// TIA Portal V17 export
// export: Created 2022-07-20T07:01:31.1393195Z, ExportSetting WithDefaults, DisplayName Totally Integrated Automation Portal, DisplayVersion V17, DisplayName TIA Portal Openness, DisplayVersion V17, DisplayName TIA Portal Version Control Interface, DisplayVersion V17, DisplayName SINAMICS Startdrive Advanced, DisplayVersion V17, DisplayName SINAMICS Startdrive G130, G150, S120, S150, SINAMICS MV, S210, DisplayVersion V17, DisplayName SINAMICS Startdrive G110M, G120, G120C, G120D, G120P, G115D, DisplayVersion V17, DisplayName STEP 7 Professional, DisplayVersion V17, DisplayName STEP 7 Safety, DisplayVersion V17, DisplayName WinCC Advanced, DisplayVersion V17
FUNCTION_BLOCK "FB10041_DetectKindOfPush"   // FB10041, LAD
{ S7_Optimized_Access := 'TRUE' }
VERSION : 0.1
// stored: AutoNumber false, IsIECCheckEnabled false, IsRetainMemResEnabled false, MemoryReserve 100, SetENOAutomatically false, UDAEnableTagReadback false
   VAR_INPUT
      Push : Bool;
   END_VAR
   VAR_OUTPUT
      ShortPushDetected : Bool;
      LongPushDetected : Bool;
   END_VAR
   VAR
      ResetCounter : Bool;
      R_TRIG_Push : R_TRIG;
      F_TRIG_Push : F_TRIG;
      FB10220_OperatingTimeCounter_Instance { S7_SetPoint := 'True'} : "FB10220_OperatingTimeCounter";
   END_VAR
BEGIN

REGION Network 1 (SCL): First Scan
   IF "FirstScan" THEN
       #ShortPushDetected := FALSE;
       #LongPushDetected := FALSE;
   END_IF;
END_REGION

REGION Network 2 (SCL)
   REGION EDGE SIGNALS
       #R_TRIG_Push(CLK := #Push);

       #F_TRIG_Push(CLK := #Push);
   END_REGION
END_REGION

REGION Network 3: Push Counter Management
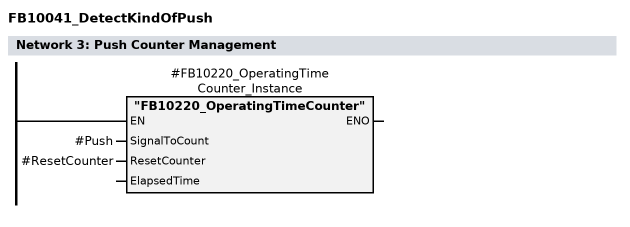
   RUNG wire#powerrail
      #FB10220_OperatingTimeCounter_Instance(SignalToCount := #Push, ResetCounter := #ResetCounter, ElapsedTime :=)
   END_RUNG
   // the same network as SCL:
   #FB10220_OperatingTimeCounter_Instance(SignalToCount := #Push, ResetCounter := #ResetCounter);   // "FB10220_OperatingTimeCounter"
END_REGION

REGION Network 4 (SCL): Kind Of Push Detection Management
   IF #R_TRIG_Push.Q THEN
       #ResetCounter := TRUE;
       #ShortPushDetected := FALSE;
       #LongPushDetected := FALSE;
   ELSIF #Push AND #FB10220_OperatingTimeCounter_Instance.ElapsedTime >= 1.0 THEN
       #ResetCounter := FALSE;
       #ShortPushDetected := FALSE;
       #LongPushDetected := TRUE;
   ELSIF #F_TRIG_Push.Q THEN
       #ResetCounter := TRUE;
       IF #FB10220_OperatingTimeCounter_Instance.ElapsedTime >= 0 AND #FB10220_OperatingTimeCounter_Instance.ElapsedTime < 1.0 THEN
           #ShortPushDetected := TRUE;
           #LongPushDetected := FALSE;
       ELSIF #FB10220_OperatingTimeCounter_Instance.ElapsedTime >= 1.0 THEN
           #ShortPushDetected := FALSE;
           #LongPushDetected := TRUE;
       END_IF;
   ELSIF NOT(#Push) THEN
       #ResetCounter := TRUE;
       #ShortPushDetected := FALSE;
       #LongPushDetected := FALSE;
   END_IF;
END_REGION
END_FUNCTION_BLOCK
